FUNCTION_BLOCK FB_WP_SchreibeDaten
VAR_INPUT
	WP_Stellung : BOOL;
END_VAR
VAR_OUTPUT
	OUT_WP_Stellung : BOOL;
END_VAR
VAR
END_VAR

OUT_WP_Stellung := WP_Stellung;

END_FUNCTION_BLOCK

(* stored: Version 1.1.0.1, ProductVersion 3.1.4024.9
   POU FB_WP_SchreibeDaten: Id {b0662140-eb81-4fd2-9d52-c33cec15be53}, SpecialFunc None *)
